// TIA Portal V17 export
// export: Created 2023-06-23T18:33:40.9538208Z, ExportSetting WithDefaults, DisplayName Totally Integrated Automation Portal, DisplayVersion V17, DisplayName TIA Portal Openness, DisplayVersion V17, DisplayName TIA Portal Version Control Interface, DisplayVersion V17, DisplayName STEP 7 Professional, DisplayVersion V17, DisplayName STEP 7 Safety, DisplayVersion V17, DisplayName WinCC Advanced / Unified PC, DisplayVersion V17
VAR_GLOBAL   // PLC tag table "26_ELR-1"
   "iELR-1" AT %I13.3 : Bool;
   "oELR-1" AT %Q12.6 : Bool;
END_VAR
